Staubli VAL3: getState.pgx

program getState()
begin
  nState=$getState()
  gotoxy(1,1)
  put("RSI state:"+toString("",nState)+"   ")
end
